// TIA Portal V16 export
// export: Created 2023-03-29T11:03:24.5102621Z, ExportSetting WithDefaults, DisplayName Totally Integrated Automation Portal, DisplayVersion V16 Update 6, DisplayName TIA Portal Version Control Interface, DisplayVersion V16 Update 2, DisplayName TIA Portal Openness, DisplayVersion V16 Update 6, DisplayName STEP 7 Professional, DisplayVersion V16 Update 6, DisplayName STEP 7 Safety, DisplayVersion V16, DisplayName WinCC Advanced, DisplayVersion V16 Update 6
FUNCTION_BLOCK "Client_ModbusTCP_sending_parameters"   // FB13, LAD
TITLE = Przesłanie parametrów sterowania
{ S7_Optimized_Access := 'TRUE' }
AUTHOR : rtecmer
VERSION : 0.1
// funkcja przkazuje parametry sterowania do PLC 1
// stored: AutoNumber true, IsIECCheckEnabled false, IsRetainMemResEnabled false, MemoryReserve 250, SetENOAutomatically false, UDAEnableTagReadback false
   VAR_IN_OUT
      modbustcp_przetwarzanie_in : Bool;
      modbustcp_przetwarzanie_out : Bool;
   END_VAR
   VAR_TEMP   // added for the SCL form of the ladder/FBD networks
      _w1 : Bool;
      _w2 : Bool;
   END_VAR
BEGIN

REGION Network 1: Inicjacja modbus po błędzie i restarcie
END_REGION

REGION Network 2
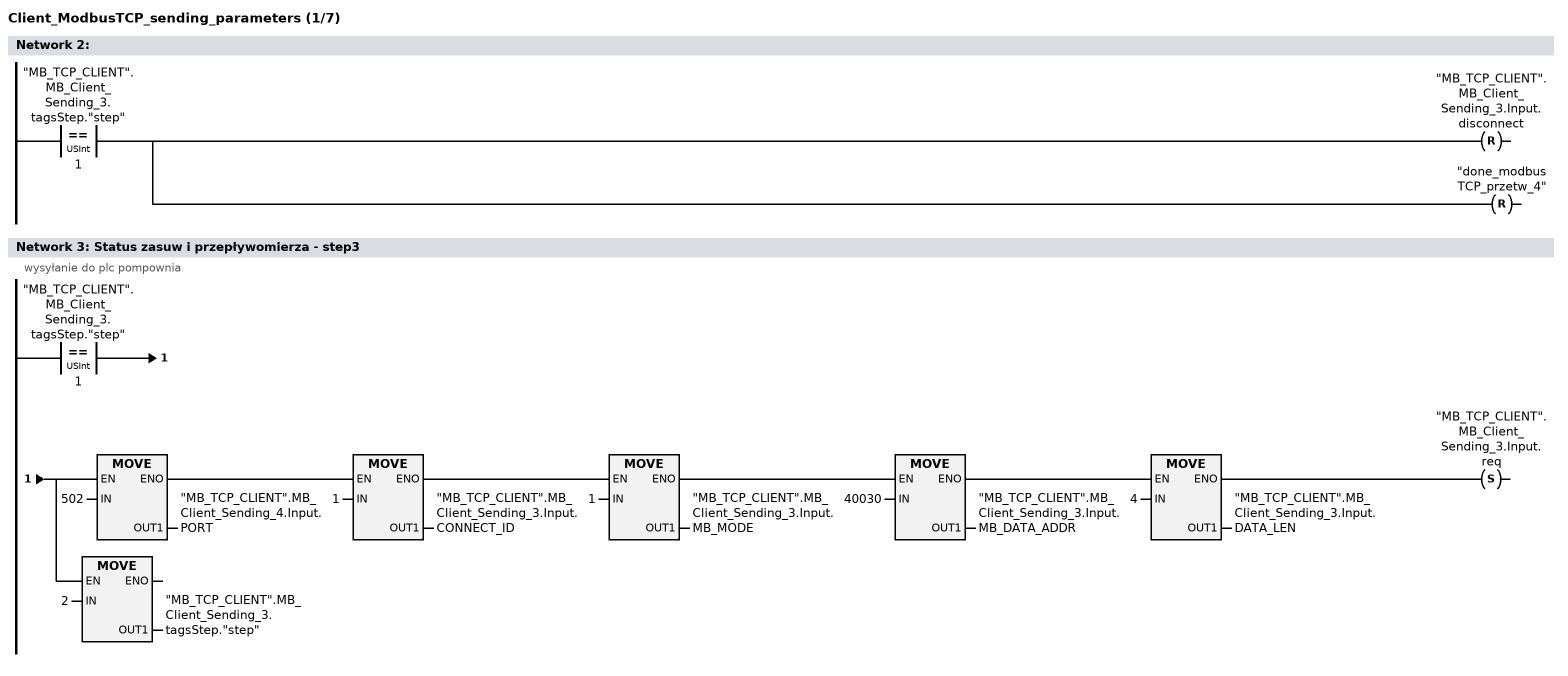
   RUNG wire#powerrail
      { S7_Templates := "SrcType := USInt" } EQ_Contact(in1 := "MB_TCP_CLIENT".MB_Client_Sending_3.tagsStep."step", in2 := 1)
      wire#w1
      R_Coil( "MB_TCP_CLIENT".MB_Client_Sending_3.Input.disconnect )
   END_RUNG
   RUNG wire#w1
      R_Coil( "done_modbusTCP_przetw_4" )
   END_RUNG
   // the same network as SCL:
   IF "MB_TCP_CLIENT".MB_Client_Sending_3.tagsStep."step" = 1 THEN
       "MB_TCP_CLIENT".MB_Client_Sending_3.Input.disconnect := FALSE;
       "done_modbusTCP_przetw_4" := FALSE;
   END_IF;
END_REGION

REGION Network 3: Status zasuw i przepływomierza - step3
   // wysyłanie do plc pompownia
   RUNG wire#powerrail
      { S7_Templates := "SrcType := USInt" } EQ_Contact(in1 := "MB_TCP_CLIENT".MB_Client_Sending_3.tagsStep."step", in2 := 1)
      wire#w1
      { S7_GenerateENO := "TRUE" } Move(in := 502, out1 => "MB_TCP_CLIENT".MB_Client_Sending_4.Input.PORT)
      { S7_GenerateENO := "TRUE" } Move(in := 1, out1 => "MB_TCP_CLIENT".MB_Client_Sending_3.Input.CONNECT_ID)
      { S7_GenerateENO := "TRUE" } Move(in := 1, out1 => "MB_TCP_CLIENT".MB_Client_Sending_3.Input.MB_MODE)
      { S7_GenerateENO := "TRUE" } Move(in := 40030, out1 => "MB_TCP_CLIENT".MB_Client_Sending_3.Input.MB_DATA_ADDR)
      { S7_GenerateENO := "TRUE" } Move(in := 4, out1 => "MB_TCP_CLIENT".MB_Client_Sending_3.Input.DATA_LEN)
      S_Coil( "MB_TCP_CLIENT".MB_Client_Sending_3.Input.req )
   END_RUNG
   RUNG wire#w1
      { S7_GenerateENO := "TRUE" } Move(in := 2, out1 => "MB_TCP_CLIENT".MB_Client_Sending_3.tagsStep."step")
   END_RUNG
   // the same network as SCL:
   // ENO of a box is taken as its EN; it also drops when the box reports an error
   IF "MB_TCP_CLIENT".MB_Client_Sending_3.tagsStep."step" = 1 THEN
       "MB_TCP_CLIENT".MB_Client_Sending_4.Input.PORT := 502;
       "MB_TCP_CLIENT".MB_Client_Sending_3.Input.CONNECT_ID := 1;
       "MB_TCP_CLIENT".MB_Client_Sending_3.Input.MB_MODE := 1;
       "MB_TCP_CLIENT".MB_Client_Sending_3.Input.MB_DATA_ADDR := 40030;
       "MB_TCP_CLIENT".MB_Client_Sending_3.Input.DATA_LEN := 4;
       "MB_TCP_CLIENT".MB_Client_Sending_3.Input.req := TRUE;
       "MB_TCP_CLIENT".MB_Client_Sending_3.tagsStep."step" := 2;
   END_IF;
END_REGION

REGION Network 4: Wysyłanie danych - step 2
   // poziom napełniania, opróżniania
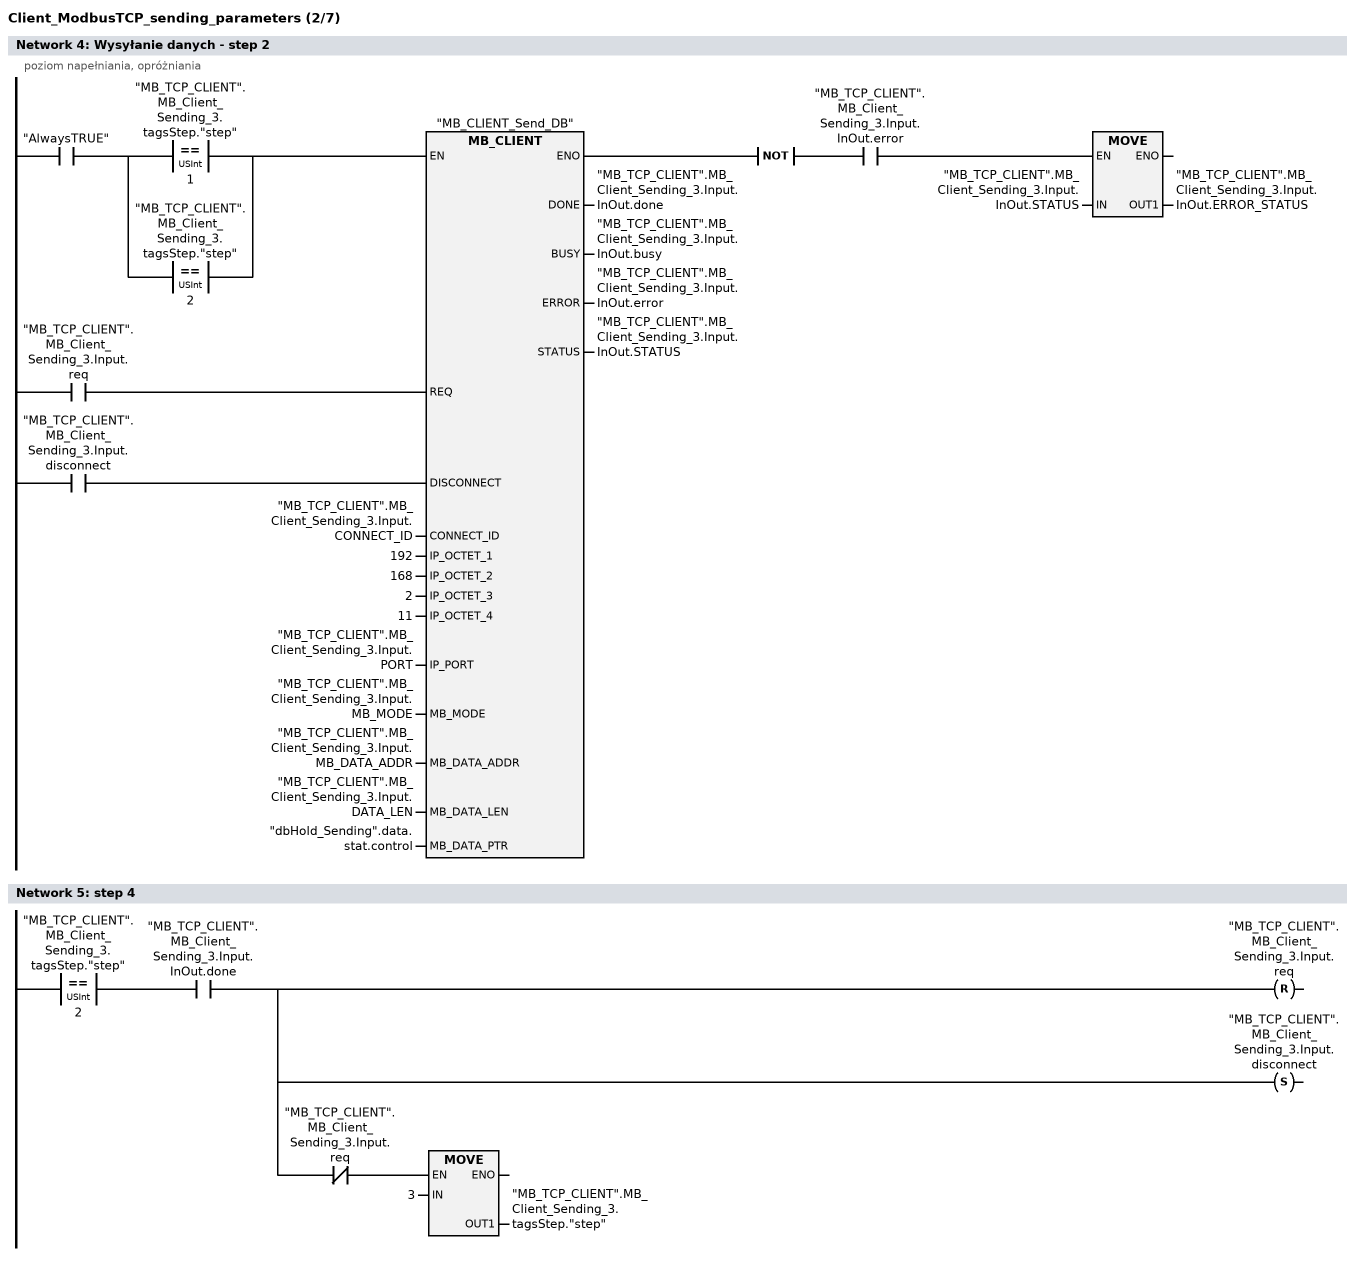
   RUNG wire#powerrail
      Contact( "AlwaysTRUE" )
      wire#w1
      { S7_Templates := "SrcType := USInt" } EQ_Contact(in1 := "MB_TCP_CLIENT".MB_Client_Sending_3.tagsStep."step", in2 := 1)
      wire#w2
      { S7_Templates := "[card1200 := 1, card1500 := 0]" } "MB_CLIENT_Send_DB".MB_CLIENT(REQ := wire#w3, DISCONNECT := wire#w4, CONNECT_ID := "MB_TCP_CLIENT".MB_Client_Sending_3.Input.CONNECT_ID, IP_OCTET_1 := 192, IP_OCTET_2 := 168, IP_OCTET_3 := 2, IP_OCTET_4 := 11, IP_PORT := "MB_TCP_CLIENT".MB_Client_Sending_3.Input.PORT, MB_MODE := "MB_TCP_CLIENT".MB_Client_Sending_3.Input.MB_MODE, MB_DATA_ADDR := "MB_TCP_CLIENT".MB_Client_Sending_3.Input.MB_DATA_ADDR, MB_DATA_LEN := "MB_TCP_CLIENT".MB_Client_Sending_3.Input.DATA_LEN, MB_DATA_PTR := "dbHold_Sending".data.stat.control, DONE => "MB_TCP_CLIENT".MB_Client_Sending_3.Input.InOut.done, BUSY => "MB_TCP_CLIENT".MB_Client_Sending_3.Input.InOut.busy, ERROR => "MB_TCP_CLIENT".MB_Client_Sending_3.Input.InOut.error, STATUS => "MB_TCP_CLIENT".MB_Client_Sending_3.Input.InOut.STATUS)
      Not()
      Contact( "MB_TCP_CLIENT".MB_Client_Sending_3.Input.InOut.error )
      Move(in := "MB_TCP_CLIENT".MB_Client_Sending_3.Input.InOut.STATUS, out1 => "MB_TCP_CLIENT".MB_Client_Sending_3.Input.InOut.ERROR_STATUS)
   END_RUNG
   RUNG wire#w1
      { S7_Templates := "SrcType := USInt" } EQ_Contact(in1 := "MB_TCP_CLIENT".MB_Client_Sending_3.tagsStep."step", in2 := 2)
   END_RUNG wire#w2
   RUNG wire#powerrail
      Contact( "MB_TCP_CLIENT".MB_Client_Sending_3.Input.req )
   END_RUNG wire#w3
   RUNG wire#powerrail
      Contact( "MB_TCP_CLIENT".MB_Client_Sending_3.Input.disconnect )
   END_RUNG wire#w4
   // the same network as SCL:
   #_w1 := "AlwaysTRUE" AND (("MB_TCP_CLIENT".MB_Client_Sending_3.tagsStep."step" = 1) OR ("MB_TCP_CLIENT".MB_Client_Sending_3.tagsStep."step" = 2));
   "MB_CLIENT_Send_DB"(EN := #_w1,   // MB_CLIENT
                       REQ := "MB_TCP_CLIENT".MB_Client_Sending_3.Input.req,
                       DISCONNECT := "MB_TCP_CLIENT".MB_Client_Sending_3.Input.disconnect,
                       CONNECT_ID := "MB_TCP_CLIENT".MB_Client_Sending_3.Input.CONNECT_ID,
                       IP_OCTET_1 := 192,
                       IP_OCTET_2 := 168,
                       IP_OCTET_3 := 2,
                       IP_OCTET_4 := 11,
                       IP_PORT := "MB_TCP_CLIENT".MB_Client_Sending_3.Input.PORT,
                       MB_MODE := "MB_TCP_CLIENT".MB_Client_Sending_3.Input.MB_MODE,
                       MB_DATA_ADDR := "MB_TCP_CLIENT".MB_Client_Sending_3.Input.MB_DATA_ADDR,
                       MB_DATA_LEN := "MB_TCP_CLIENT".MB_Client_Sending_3.Input.DATA_LEN,
                       MB_DATA_PTR := "dbHold_Sending".data.stat.control,
                       DONE => "MB_TCP_CLIENT".MB_Client_Sending_3.Input.InOut.done,
                       BUSY => "MB_TCP_CLIENT".MB_Client_Sending_3.Input.InOut.busy,
                       ERROR => "MB_TCP_CLIENT".MB_Client_Sending_3.Input.InOut.error,
                       STATUS => "MB_TCP_CLIENT".MB_Client_Sending_3.Input.InOut.STATUS,
                       ENO => #_w2);
   IF NOT #_w2 AND "MB_TCP_CLIENT".MB_Client_Sending_3.Input.InOut.error THEN
       "MB_TCP_CLIENT".MB_Client_Sending_3.Input.InOut.ERROR_STATUS := "MB_TCP_CLIENT".MB_Client_Sending_3.Input.InOut.STATUS;
   END_IF;
END_REGION

REGION Network 5: step 4
   RUNG wire#powerrail
      { S7_Templates := "SrcType := USInt" } EQ_Contact(in1 := "MB_TCP_CLIENT".MB_Client_Sending_3.tagsStep."step", in2 := 2)
      Contact( "MB_TCP_CLIENT".MB_Client_Sending_3.Input.InOut.done )
      wire#w1
      R_Coil( "MB_TCP_CLIENT".MB_Client_Sending_3.Input.req )
   END_RUNG
   RUNG wire#w1
      S_Coil( "MB_TCP_CLIENT".MB_Client_Sending_3.Input.disconnect )
   END_RUNG
   RUNG wire#w1
      I_Contact( "MB_TCP_CLIENT".MB_Client_Sending_3.Input.req )
      Move(in := 3, out1 => "MB_TCP_CLIENT".MB_Client_Sending_3.tagsStep."step")
   END_RUNG
   // the same network as SCL:
   #_w1 := ("MB_TCP_CLIENT".MB_Client_Sending_3.tagsStep."step" = 2) AND "MB_TCP_CLIENT".MB_Client_Sending_3.Input.InOut.done;
   IF #_w1 THEN
       "MB_TCP_CLIENT".MB_Client_Sending_3.Input.req := FALSE;
       "MB_TCP_CLIENT".MB_Client_Sending_3.Input.disconnect := TRUE;
   END_IF;
   IF #_w1 AND NOT "MB_TCP_CLIENT".MB_Client_Sending_3.Input.req THEN
       "MB_TCP_CLIENT".MB_Client_Sending_3.tagsStep."step" := 3;
   END_IF;
END_REGION

REGION Network 6
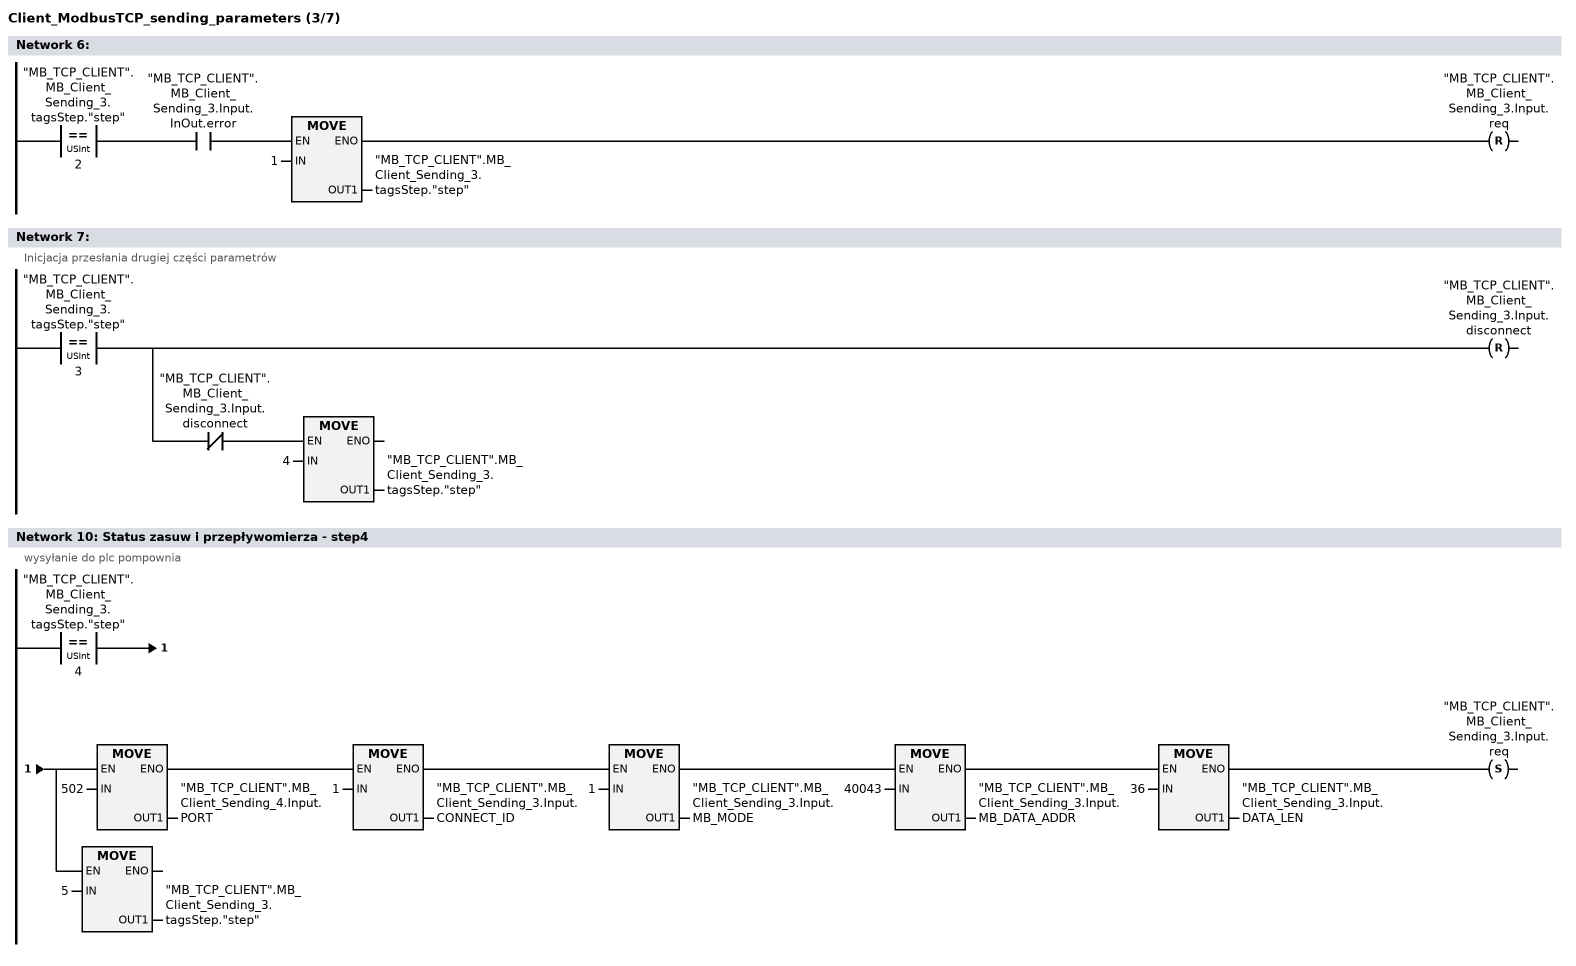
   RUNG wire#powerrail
      { S7_Templates := "SrcType := USInt" } EQ_Contact(in1 := "MB_TCP_CLIENT".MB_Client_Sending_3.tagsStep."step", in2 := 2)
      Contact( "MB_TCP_CLIENT".MB_Client_Sending_3.Input.InOut.error )
      Move(in := 1, out1 => "MB_TCP_CLIENT".MB_Client_Sending_3.tagsStep."step")
      R_Coil( "MB_TCP_CLIENT".MB_Client_Sending_3.Input.req )
   END_RUNG
   // the same network as SCL:
   #_w1 := ("MB_TCP_CLIENT".MB_Client_Sending_3.tagsStep."step" = 2) AND "MB_TCP_CLIENT".MB_Client_Sending_3.Input.InOut.error;
   IF #_w1 THEN
       "MB_TCP_CLIENT".MB_Client_Sending_3.tagsStep."step" := 1;
       "MB_TCP_CLIENT".MB_Client_Sending_3.Input.req := FALSE;
   END_IF;
END_REGION

REGION Network 7
   // Inicjacja przesłania drugiej części parametrów
   RUNG wire#powerrail
      { S7_Templates := "SrcType := USInt" } EQ_Contact(in1 := "MB_TCP_CLIENT".MB_Client_Sending_3.tagsStep."step", in2 := 3)
      wire#w1
      R_Coil( "MB_TCP_CLIENT".MB_Client_Sending_3.Input.disconnect )
   END_RUNG
   RUNG wire#w1
      I_Contact( "MB_TCP_CLIENT".MB_Client_Sending_3.Input.disconnect )
      Move(in := 4, out1 => "MB_TCP_CLIENT".MB_Client_Sending_3.tagsStep."step")
   END_RUNG
   // the same network as SCL:
   #_w1 := "MB_TCP_CLIENT".MB_Client_Sending_3.tagsStep."step" = 3;
   IF #_w1 THEN "MB_TCP_CLIENT".MB_Client_Sending_3.Input.disconnect := FALSE; END_IF;
   IF #_w1 AND NOT "MB_TCP_CLIENT".MB_Client_Sending_3.Input.disconnect THEN
       "MB_TCP_CLIENT".MB_Client_Sending_3.tagsStep."step" := 4;
   END_IF;
END_REGION

REGION Network 10: Status zasuw i przepływomierza - step4
   // wysyłanie do plc pompownia
   RUNG wire#powerrail
      { S7_Templates := "SrcType := USInt" } EQ_Contact(in1 := "MB_TCP_CLIENT".MB_Client_Sending_3.tagsStep."step", in2 := 4)
      wire#w1
      { S7_GenerateENO := "TRUE" } Move(in := 502, out1 => "MB_TCP_CLIENT".MB_Client_Sending_4.Input.PORT)
      { S7_GenerateENO := "TRUE" } Move(in := 1, out1 => "MB_TCP_CLIENT".MB_Client_Sending_3.Input.CONNECT_ID)
      { S7_GenerateENO := "TRUE" } Move(in := 1, out1 => "MB_TCP_CLIENT".MB_Client_Sending_3.Input.MB_MODE)
      { S7_GenerateENO := "TRUE" } Move(in := 40043, out1 => "MB_TCP_CLIENT".MB_Client_Sending_3.Input.MB_DATA_ADDR)
      { S7_GenerateENO := "TRUE" } Move(in := 36, out1 => "MB_TCP_CLIENT".MB_Client_Sending_3.Input.DATA_LEN)
      S_Coil( "MB_TCP_CLIENT".MB_Client_Sending_3.Input.req )
   END_RUNG
   RUNG wire#w1
      { S7_GenerateENO := "TRUE" } Move(in := 5, out1 => "MB_TCP_CLIENT".MB_Client_Sending_3.tagsStep."step")
   END_RUNG
   // the same network as SCL:
   // ENO of a box is taken as its EN; it also drops when the box reports an error
   IF "MB_TCP_CLIENT".MB_Client_Sending_3.tagsStep."step" = 4 THEN
       "MB_TCP_CLIENT".MB_Client_Sending_4.Input.PORT := 502;
       "MB_TCP_CLIENT".MB_Client_Sending_3.Input.CONNECT_ID := 1;
       "MB_TCP_CLIENT".MB_Client_Sending_3.Input.MB_MODE := 1;
       "MB_TCP_CLIENT".MB_Client_Sending_3.Input.MB_DATA_ADDR := 40043;
       "MB_TCP_CLIENT".MB_Client_Sending_3.Input.DATA_LEN := 36;
       "MB_TCP_CLIENT".MB_Client_Sending_3.Input.req := TRUE;
       "MB_TCP_CLIENT".MB_Client_Sending_3.tagsStep."step" := 5;
   END_IF;
END_REGION

REGION Network 11: Wysyłanie danych - step 2
   // poziom napełniania, opróżniania
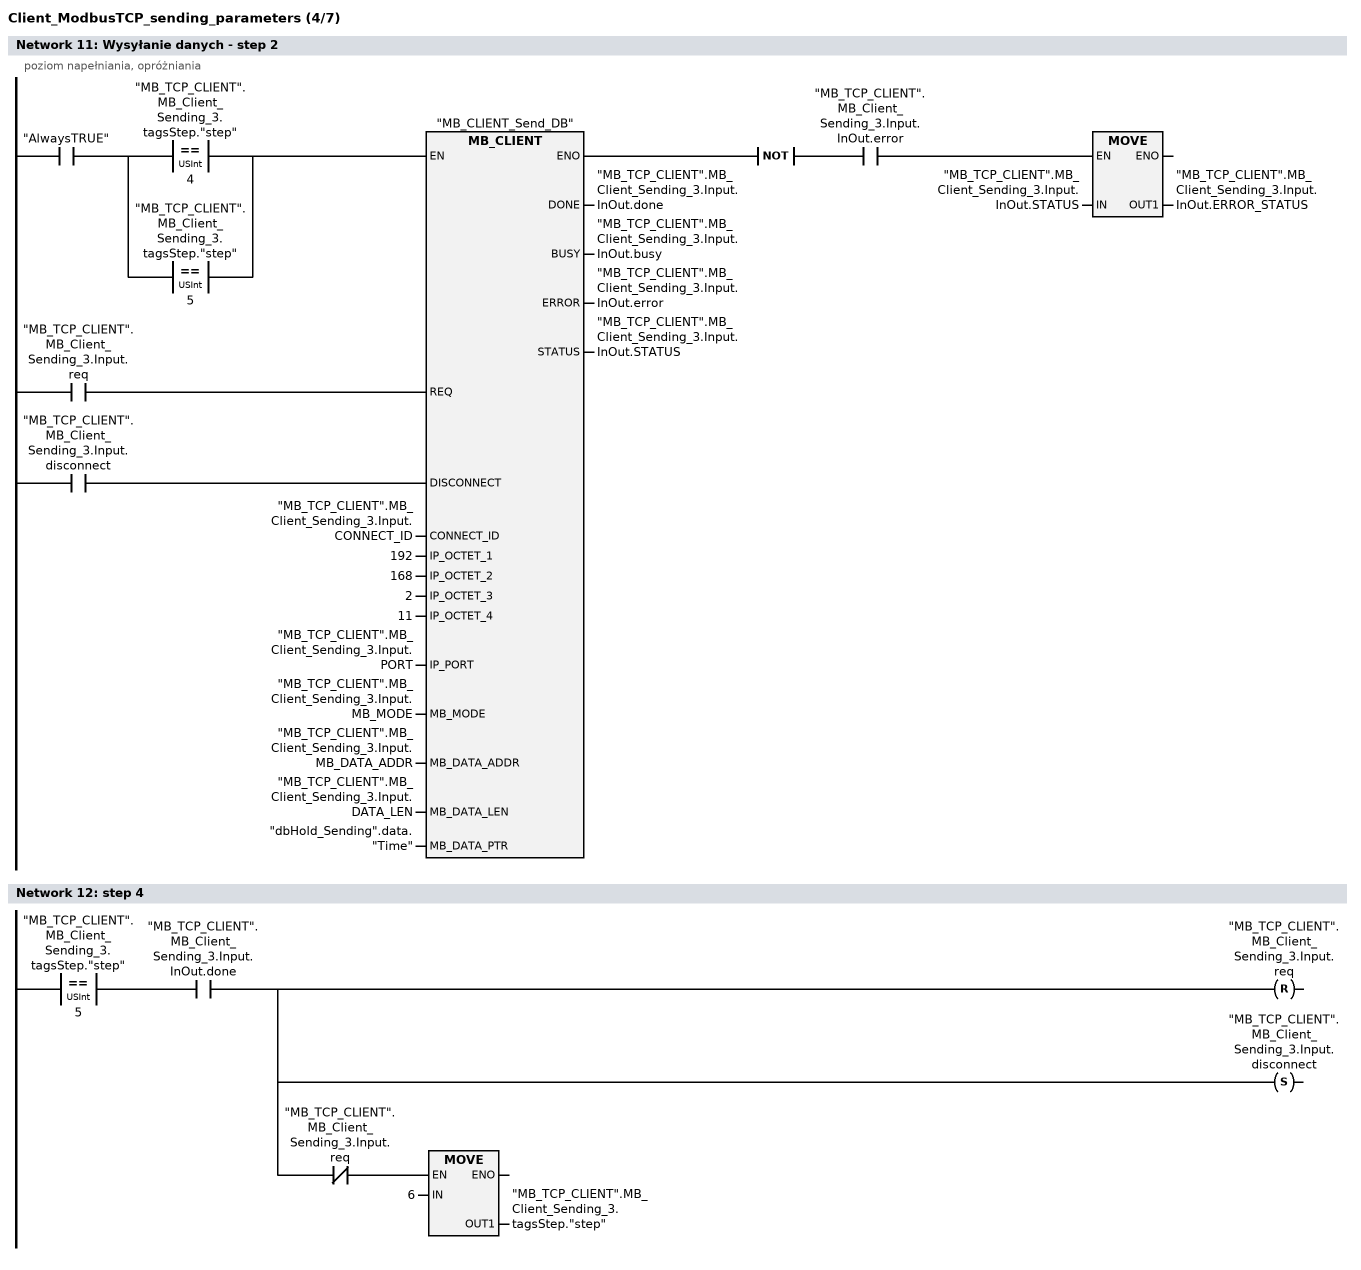
   RUNG wire#powerrail
      Contact( "AlwaysTRUE" )
      wire#w1
      { S7_Templates := "SrcType := USInt" } EQ_Contact(in1 := "MB_TCP_CLIENT".MB_Client_Sending_3.tagsStep."step", in2 := 4)
      wire#w2
      { S7_Templates := "[card1200 := 1, card1500 := 0]" } "MB_CLIENT_Send_DB".MB_CLIENT(REQ := wire#w3, DISCONNECT := wire#w4, CONNECT_ID := "MB_TCP_CLIENT".MB_Client_Sending_3.Input.CONNECT_ID, IP_OCTET_1 := 192, IP_OCTET_2 := 168, IP_OCTET_3 := 2, IP_OCTET_4 := 11, IP_PORT := "MB_TCP_CLIENT".MB_Client_Sending_3.Input.PORT, MB_MODE := "MB_TCP_CLIENT".MB_Client_Sending_3.Input.MB_MODE, MB_DATA_ADDR := "MB_TCP_CLIENT".MB_Client_Sending_3.Input.MB_DATA_ADDR, MB_DATA_LEN := "MB_TCP_CLIENT".MB_Client_Sending_3.Input.DATA_LEN, MB_DATA_PTR := "dbHold_Sending".data."Time", DONE => "MB_TCP_CLIENT".MB_Client_Sending_3.Input.InOut.done, BUSY => "MB_TCP_CLIENT".MB_Client_Sending_3.Input.InOut.busy, ERROR => "MB_TCP_CLIENT".MB_Client_Sending_3.Input.InOut.error, STATUS => "MB_TCP_CLIENT".MB_Client_Sending_3.Input.InOut.STATUS)
      Not()
      Contact( "MB_TCP_CLIENT".MB_Client_Sending_3.Input.InOut.error )
      Move(in := "MB_TCP_CLIENT".MB_Client_Sending_3.Input.InOut.STATUS, out1 => "MB_TCP_CLIENT".MB_Client_Sending_3.Input.InOut.ERROR_STATUS)
   END_RUNG
   RUNG wire#w1
      { S7_Templates := "SrcType := USInt" } EQ_Contact(in1 := "MB_TCP_CLIENT".MB_Client_Sending_3.tagsStep."step", in2 := 5)
   END_RUNG wire#w2
   RUNG wire#powerrail
      Contact( "MB_TCP_CLIENT".MB_Client_Sending_3.Input.req )
   END_RUNG wire#w3
   RUNG wire#powerrail
      Contact( "MB_TCP_CLIENT".MB_Client_Sending_3.Input.disconnect )
   END_RUNG wire#w4
   // the same network as SCL:
   #_w1 := "AlwaysTRUE" AND (("MB_TCP_CLIENT".MB_Client_Sending_3.tagsStep."step" = 4) OR ("MB_TCP_CLIENT".MB_Client_Sending_3.tagsStep."step" = 5));
   "MB_CLIENT_Send_DB"(EN := #_w1,   // MB_CLIENT
                       REQ := "MB_TCP_CLIENT".MB_Client_Sending_3.Input.req,
                       DISCONNECT := "MB_TCP_CLIENT".MB_Client_Sending_3.Input.disconnect,
                       CONNECT_ID := "MB_TCP_CLIENT".MB_Client_Sending_3.Input.CONNECT_ID,
                       IP_OCTET_1 := 192,
                       IP_OCTET_2 := 168,
                       IP_OCTET_3 := 2,
                       IP_OCTET_4 := 11,
                       IP_PORT := "MB_TCP_CLIENT".MB_Client_Sending_3.Input.PORT,
                       MB_MODE := "MB_TCP_CLIENT".MB_Client_Sending_3.Input.MB_MODE,
                       MB_DATA_ADDR := "MB_TCP_CLIENT".MB_Client_Sending_3.Input.MB_DATA_ADDR,
                       MB_DATA_LEN := "MB_TCP_CLIENT".MB_Client_Sending_3.Input.DATA_LEN,
                       MB_DATA_PTR := "dbHold_Sending".data."Time",
                       DONE => "MB_TCP_CLIENT".MB_Client_Sending_3.Input.InOut.done,
                       BUSY => "MB_TCP_CLIENT".MB_Client_Sending_3.Input.InOut.busy,
                       ERROR => "MB_TCP_CLIENT".MB_Client_Sending_3.Input.InOut.error,
                       STATUS => "MB_TCP_CLIENT".MB_Client_Sending_3.Input.InOut.STATUS,
                       ENO => #_w2);
   IF NOT #_w2 AND "MB_TCP_CLIENT".MB_Client_Sending_3.Input.InOut.error THEN
       "MB_TCP_CLIENT".MB_Client_Sending_3.Input.InOut.ERROR_STATUS := "MB_TCP_CLIENT".MB_Client_Sending_3.Input.InOut.STATUS;
   END_IF;
END_REGION

REGION Network 12: step 4
   RUNG wire#powerrail
      { S7_Templates := "SrcType := USInt" } EQ_Contact(in1 := "MB_TCP_CLIENT".MB_Client_Sending_3.tagsStep."step", in2 := 5)
      Contact( "MB_TCP_CLIENT".MB_Client_Sending_3.Input.InOut.done )
      wire#w1
      R_Coil( "MB_TCP_CLIENT".MB_Client_Sending_3.Input.req )
   END_RUNG
   RUNG wire#w1
      S_Coil( "MB_TCP_CLIENT".MB_Client_Sending_3.Input.disconnect )
   END_RUNG
   RUNG wire#w1
      I_Contact( "MB_TCP_CLIENT".MB_Client_Sending_3.Input.req )
      Move(in := 6, out1 => "MB_TCP_CLIENT".MB_Client_Sending_3.tagsStep."step")
   END_RUNG
   // the same network as SCL:
   #_w1 := ("MB_TCP_CLIENT".MB_Client_Sending_3.tagsStep."step" = 5) AND "MB_TCP_CLIENT".MB_Client_Sending_3.Input.InOut.done;
   IF #_w1 THEN
       "MB_TCP_CLIENT".MB_Client_Sending_3.Input.req := FALSE;
       "MB_TCP_CLIENT".MB_Client_Sending_3.Input.disconnect := TRUE;
   END_IF;
   IF #_w1 AND NOT "MB_TCP_CLIENT".MB_Client_Sending_3.Input.req THEN
       "MB_TCP_CLIENT".MB_Client_Sending_3.tagsStep."step" := 6;
   END_IF;
END_REGION

REGION Network 13
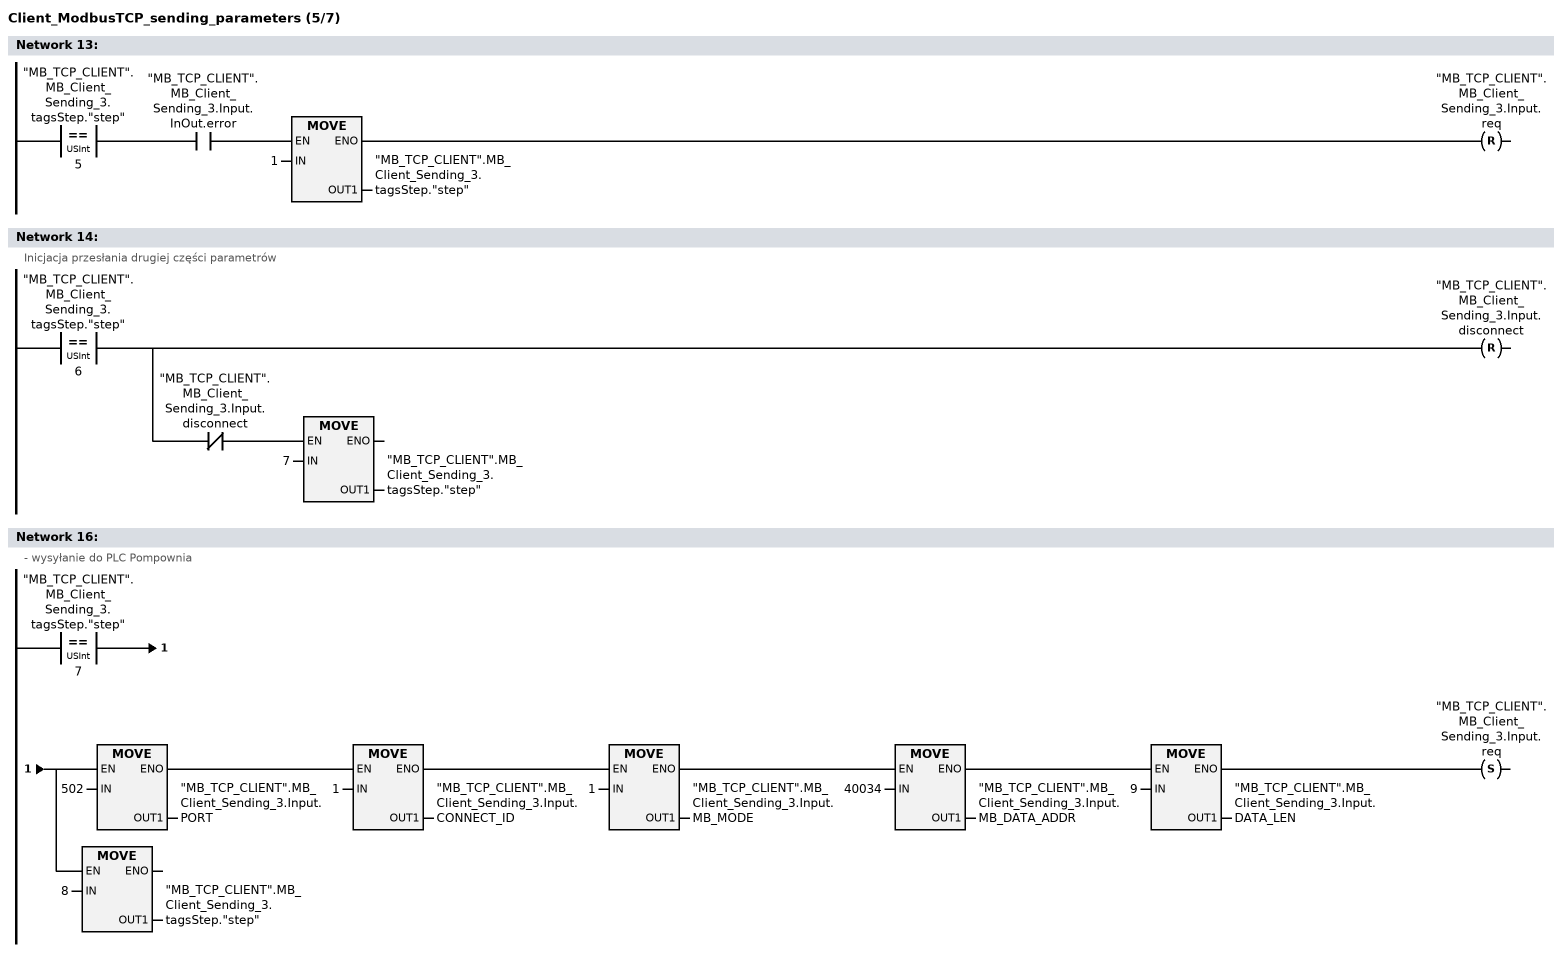
   RUNG wire#powerrail
      { S7_Templates := "SrcType := USInt" } EQ_Contact(in1 := "MB_TCP_CLIENT".MB_Client_Sending_3.tagsStep."step", in2 := 5)
      Contact( "MB_TCP_CLIENT".MB_Client_Sending_3.Input.InOut.error )
      Move(in := 1, out1 => "MB_TCP_CLIENT".MB_Client_Sending_3.tagsStep."step")
      R_Coil( "MB_TCP_CLIENT".MB_Client_Sending_3.Input.req )
   END_RUNG
   // the same network as SCL:
   #_w1 := ("MB_TCP_CLIENT".MB_Client_Sending_3.tagsStep."step" = 5) AND "MB_TCP_CLIENT".MB_Client_Sending_3.Input.InOut.error;
   IF #_w1 THEN
       "MB_TCP_CLIENT".MB_Client_Sending_3.tagsStep."step" := 1;
       "MB_TCP_CLIENT".MB_Client_Sending_3.Input.req := FALSE;
   END_IF;
END_REGION

REGION Network 14
   // Inicjacja przesłania drugiej części parametrów
   RUNG wire#powerrail
      { S7_Templates := "SrcType := USInt" } EQ_Contact(in1 := "MB_TCP_CLIENT".MB_Client_Sending_3.tagsStep."step", in2 := 6)
      wire#w1
      R_Coil( "MB_TCP_CLIENT".MB_Client_Sending_3.Input.disconnect )
   END_RUNG
   RUNG wire#w1
      I_Contact( "MB_TCP_CLIENT".MB_Client_Sending_3.Input.disconnect )
      Move(in := 7, out1 => "MB_TCP_CLIENT".MB_Client_Sending_3.tagsStep."step")
   END_RUNG
   // the same network as SCL:
   #_w1 := "MB_TCP_CLIENT".MB_Client_Sending_3.tagsStep."step" = 6;
   IF #_w1 THEN "MB_TCP_CLIENT".MB_Client_Sending_3.Input.disconnect := FALSE; END_IF;
   IF #_w1 AND NOT "MB_TCP_CLIENT".MB_Client_Sending_3.Input.disconnect THEN
       "MB_TCP_CLIENT".MB_Client_Sending_3.tagsStep."step" := 7;
   END_IF;
END_REGION

REGION Network 16
   // - wysyłanie do PLC Pompownia
   RUNG wire#powerrail
      { S7_Templates := "SrcType := USInt" } EQ_Contact(in1 := "MB_TCP_CLIENT".MB_Client_Sending_3.tagsStep."step", in2 := 7)
      wire#w1
      { S7_GenerateENO := "TRUE" } Move(in := 502, out1 => "MB_TCP_CLIENT".MB_Client_Sending_3.Input.PORT)
      { S7_GenerateENO := "TRUE" } Move(in := 1, out1 => "MB_TCP_CLIENT".MB_Client_Sending_3.Input.CONNECT_ID)
      { S7_GenerateENO := "TRUE" } Move(in := 1, out1 => "MB_TCP_CLIENT".MB_Client_Sending_3.Input.MB_MODE)
      { S7_GenerateENO := "TRUE" } Move(in := 40034, out1 => "MB_TCP_CLIENT".MB_Client_Sending_3.Input.MB_DATA_ADDR)
      { S7_GenerateENO := "TRUE" } Move(in := 9, out1 => "MB_TCP_CLIENT".MB_Client_Sending_3.Input.DATA_LEN)
      S_Coil( "MB_TCP_CLIENT".MB_Client_Sending_3.Input.req )
   END_RUNG
   RUNG wire#w1
      { S7_GenerateENO := "TRUE" } Move(in := 8, out1 => "MB_TCP_CLIENT".MB_Client_Sending_3.tagsStep."step")
   END_RUNG
   // the same network as SCL:
   // ENO of a box is taken as its EN; it also drops when the box reports an error
   IF "MB_TCP_CLIENT".MB_Client_Sending_3.tagsStep."step" = 7 THEN
       "MB_TCP_CLIENT".MB_Client_Sending_3.Input.PORT := 502;
       "MB_TCP_CLIENT".MB_Client_Sending_3.Input.CONNECT_ID := 1;
       "MB_TCP_CLIENT".MB_Client_Sending_3.Input.MB_MODE := 1;
       "MB_TCP_CLIENT".MB_Client_Sending_3.Input.MB_DATA_ADDR := 40034;
       "MB_TCP_CLIENT".MB_Client_Sending_3.Input.DATA_LEN := 9;
       "MB_TCP_CLIENT".MB_Client_Sending_3.Input.req := TRUE;
       "MB_TCP_CLIENT".MB_Client_Sending_3.tagsStep."step" := 8;
   END_IF;
END_REGION

REGION Network 17: Wysyłanie danych - step 2
   // Analogi
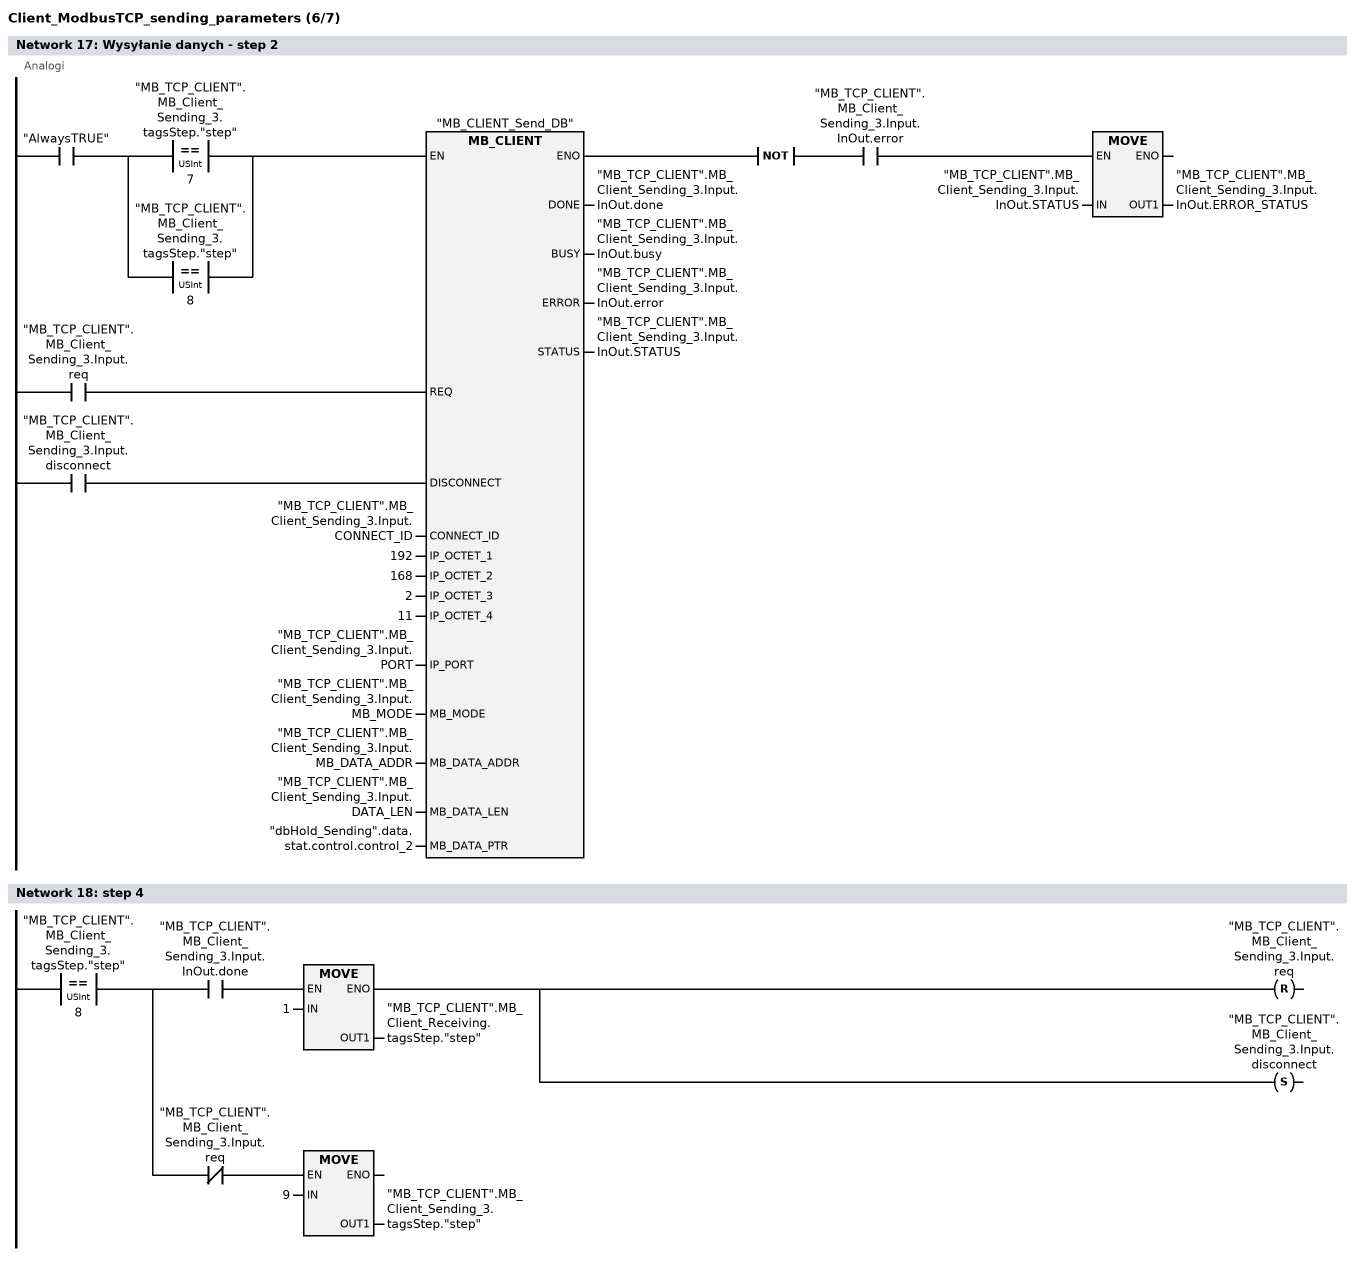
   RUNG wire#powerrail
      Contact( "AlwaysTRUE" )
      wire#w1
      { S7_Templates := "SrcType := USInt" } EQ_Contact(in1 := "MB_TCP_CLIENT".MB_Client_Sending_3.tagsStep."step", in2 := 7)
      wire#w2
      { S7_Templates := "[card1200 := 1, card1500 := 0]" } "MB_CLIENT_Send_DB".MB_CLIENT(REQ := wire#w3, DISCONNECT := wire#w4, CONNECT_ID := "MB_TCP_CLIENT".MB_Client_Sending_3.Input.CONNECT_ID, IP_OCTET_1 := 192, IP_OCTET_2 := 168, IP_OCTET_3 := 2, IP_OCTET_4 := 11, IP_PORT := "MB_TCP_CLIENT".MB_Client_Sending_3.Input.PORT, MB_MODE := "MB_TCP_CLIENT".MB_Client_Sending_3.Input.MB_MODE, MB_DATA_ADDR := "MB_TCP_CLIENT".MB_Client_Sending_3.Input.MB_DATA_ADDR, MB_DATA_LEN := "MB_TCP_CLIENT".MB_Client_Sending_3.Input.DATA_LEN, MB_DATA_PTR := "dbHold_Sending".data.stat.control.control_2, DONE => "MB_TCP_CLIENT".MB_Client_Sending_3.Input.InOut.done, BUSY => "MB_TCP_CLIENT".MB_Client_Sending_3.Input.InOut.busy, ERROR => "MB_TCP_CLIENT".MB_Client_Sending_3.Input.InOut.error, STATUS => "MB_TCP_CLIENT".MB_Client_Sending_3.Input.InOut.STATUS)
      Not()
      Contact( "MB_TCP_CLIENT".MB_Client_Sending_3.Input.InOut.error )
      Move(in := "MB_TCP_CLIENT".MB_Client_Sending_3.Input.InOut.STATUS, out1 => "MB_TCP_CLIENT".MB_Client_Sending_3.Input.InOut.ERROR_STATUS)
   END_RUNG
   RUNG wire#w1
      { S7_Templates := "SrcType := USInt" } EQ_Contact(in1 := "MB_TCP_CLIENT".MB_Client_Sending_3.tagsStep."step", in2 := 8)
   END_RUNG wire#w2
   RUNG wire#powerrail
      Contact( "MB_TCP_CLIENT".MB_Client_Sending_3.Input.req )
   END_RUNG wire#w3
   RUNG wire#powerrail
      Contact( "MB_TCP_CLIENT".MB_Client_Sending_3.Input.disconnect )
   END_RUNG wire#w4
   // the same network as SCL:
   #_w1 := "AlwaysTRUE" AND (("MB_TCP_CLIENT".MB_Client_Sending_3.tagsStep."step" = 7) OR ("MB_TCP_CLIENT".MB_Client_Sending_3.tagsStep."step" = 8));
   "MB_CLIENT_Send_DB"(EN := #_w1,   // MB_CLIENT
                       REQ := "MB_TCP_CLIENT".MB_Client_Sending_3.Input.req,
                       DISCONNECT := "MB_TCP_CLIENT".MB_Client_Sending_3.Input.disconnect,
                       CONNECT_ID := "MB_TCP_CLIENT".MB_Client_Sending_3.Input.CONNECT_ID,
                       IP_OCTET_1 := 192,
                       IP_OCTET_2 := 168,
                       IP_OCTET_3 := 2,
                       IP_OCTET_4 := 11,
                       IP_PORT := "MB_TCP_CLIENT".MB_Client_Sending_3.Input.PORT,
                       MB_MODE := "MB_TCP_CLIENT".MB_Client_Sending_3.Input.MB_MODE,
                       MB_DATA_ADDR := "MB_TCP_CLIENT".MB_Client_Sending_3.Input.MB_DATA_ADDR,
                       MB_DATA_LEN := "MB_TCP_CLIENT".MB_Client_Sending_3.Input.DATA_LEN,
                       MB_DATA_PTR := "dbHold_Sending".data.stat.control.control_2,
                       DONE => "MB_TCP_CLIENT".MB_Client_Sending_3.Input.InOut.done,
                       BUSY => "MB_TCP_CLIENT".MB_Client_Sending_3.Input.InOut.busy,
                       ERROR => "MB_TCP_CLIENT".MB_Client_Sending_3.Input.InOut.error,
                       STATUS => "MB_TCP_CLIENT".MB_Client_Sending_3.Input.InOut.STATUS,
                       ENO => #_w2);
   IF NOT #_w2 AND "MB_TCP_CLIENT".MB_Client_Sending_3.Input.InOut.error THEN
       "MB_TCP_CLIENT".MB_Client_Sending_3.Input.InOut.ERROR_STATUS := "MB_TCP_CLIENT".MB_Client_Sending_3.Input.InOut.STATUS;
   END_IF;
END_REGION

REGION Network 18: step 4
   RUNG wire#powerrail
      { S7_Templates := "SrcType := USInt" } EQ_Contact(in1 := "MB_TCP_CLIENT".MB_Client_Sending_3.tagsStep."step", in2 := 8)
      wire#w1
      Contact( "MB_TCP_CLIENT".MB_Client_Sending_3.Input.InOut.done )
      Move(in := 1, out1 => "MB_TCP_CLIENT".MB_Client_Receiving.tagsStep."step")
      wire#w2
      R_Coil( "MB_TCP_CLIENT".MB_Client_Sending_3.Input.req )
   END_RUNG
   RUNG wire#w2
      S_Coil( "MB_TCP_CLIENT".MB_Client_Sending_3.Input.disconnect )
   END_RUNG
   RUNG wire#w1
      I_Contact( "MB_TCP_CLIENT".MB_Client_Sending_3.Input.req )
      Move(in := 9, out1 => "MB_TCP_CLIENT".MB_Client_Sending_3.tagsStep."step")
   END_RUNG
   // the same network as SCL:
   #_w1 := "MB_TCP_CLIENT".MB_Client_Sending_3.tagsStep."step" = 8;
   IF #_w1 AND "MB_TCP_CLIENT".MB_Client_Sending_3.Input.InOut.done THEN
       "MB_TCP_CLIENT".MB_Client_Receiving.tagsStep."step" := 1;
       "MB_TCP_CLIENT".MB_Client_Sending_3.Input.req := FALSE;
       "MB_TCP_CLIENT".MB_Client_Sending_3.Input.disconnect := TRUE;
   END_IF;
   IF #_w1 AND NOT "MB_TCP_CLIENT".MB_Client_Sending_3.Input.req THEN
       "MB_TCP_CLIENT".MB_Client_Sending_3.tagsStep."step" := 9;
   END_IF;
END_REGION

REGION Network 19
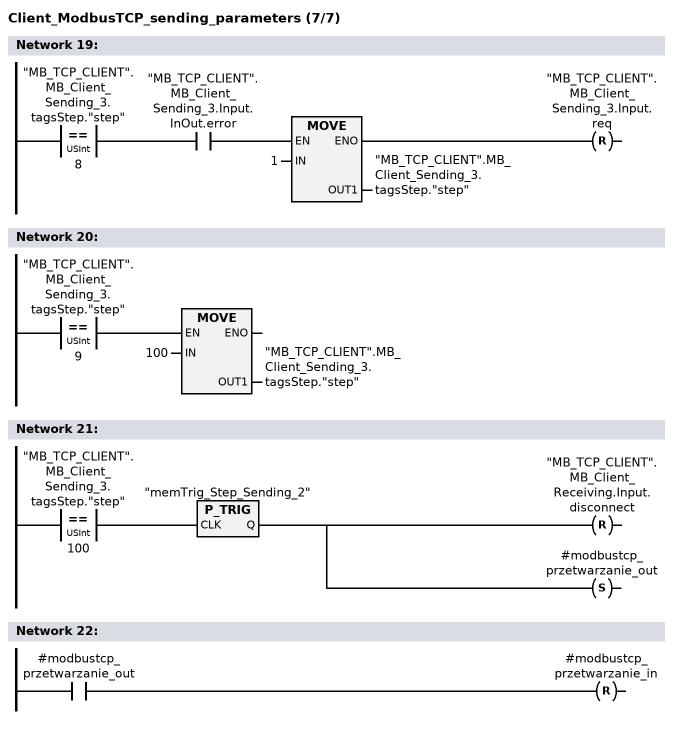
   RUNG wire#powerrail
      { S7_Templates := "SrcType := USInt" } EQ_Contact(in1 := "MB_TCP_CLIENT".MB_Client_Sending_3.tagsStep."step", in2 := 8)
      Contact( "MB_TCP_CLIENT".MB_Client_Sending_3.Input.InOut.error )
      Move(in := 1, out1 => "MB_TCP_CLIENT".MB_Client_Sending_3.tagsStep."step")
      R_Coil( "MB_TCP_CLIENT".MB_Client_Sending_3.Input.req )
   END_RUNG
   // the same network as SCL:
   #_w1 := ("MB_TCP_CLIENT".MB_Client_Sending_3.tagsStep."step" = 8) AND "MB_TCP_CLIENT".MB_Client_Sending_3.Input.InOut.error;
   IF #_w1 THEN
       "MB_TCP_CLIENT".MB_Client_Sending_3.tagsStep."step" := 1;
       "MB_TCP_CLIENT".MB_Client_Sending_3.Input.req := FALSE;
   END_IF;
END_REGION

REGION Network 20
   RUNG wire#powerrail
      { S7_Templates := "SrcType := USInt" } EQ_Contact(in1 := "MB_TCP_CLIENT".MB_Client_Sending_3.tagsStep."step", in2 := 9)
      Move(in := 100, out1 => "MB_TCP_CLIENT".MB_Client_Sending_3.tagsStep."step")
   END_RUNG
   // the same network as SCL:
   IF "MB_TCP_CLIENT".MB_Client_Sending_3.tagsStep."step" = 9 THEN
       "MB_TCP_CLIENT".MB_Client_Sending_3.tagsStep."step" := 100;
   END_IF;
END_REGION

REGION Network 21
   RUNG wire#powerrail
      { S7_Templates := "SrcType := USInt" } EQ_Contact(in1 := "MB_TCP_CLIENT".MB_Client_Sending_3.tagsStep."step", in2 := 100)
      P_Trig( "memTrig_Step_Sending_2" )
      wire#w1
      R_Coil( "MB_TCP_CLIENT".MB_Client_Receiving.Input.disconnect )
   END_RUNG
   RUNG wire#w1
      S_Coil( #modbustcp_przetwarzanie_out )
   END_RUNG
   // the same network as SCL:
   #_w1 := "MB_TCP_CLIENT".MB_Client_Sending_3.tagsStep."step" = 100;
   #_w2 := #_w1 AND NOT "memTrig_Step_Sending_2";   // rising edge
   "memTrig_Step_Sending_2" := #_w1;
   IF #_w2 THEN
       "MB_TCP_CLIENT".MB_Client_Receiving.Input.disconnect := FALSE;
       #modbustcp_przetwarzanie_out := TRUE;
   END_IF;
END_REGION

REGION Network 22
   RUNG wire#powerrail
      Contact( #modbustcp_przetwarzanie_out )
      R_Coil( #modbustcp_przetwarzanie_in )
   END_RUNG
   // the same network as SCL:
   IF #modbustcp_przetwarzanie_out THEN #modbustcp_przetwarzanie_in := FALSE; END_IF;
END_REGION
END_FUNCTION_BLOCK
